(* PLC project Unnamed, Unknown Unnamed 1 *)
(* stored: creationDateTime 2022-08-16T15:49:17, modificationDateTime 2025-06-02T17:15:43 *)

PROGRAM Blink
  VAR
    blink_led : BOOL;
    TON0 : TON;
    TOF0 : TOF;
  END_VAR

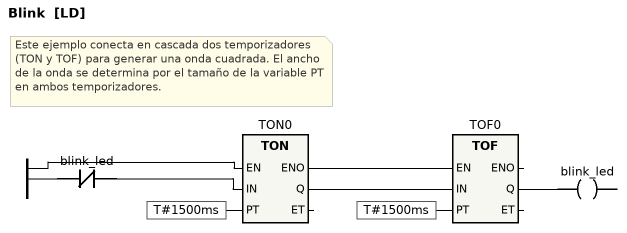
(* LD diagram, written out as Structured Text *)
(* Este ejemplo conecta en cascada dos temporizadores (TON y TOF) para generar una onda cuadrada. El ancho de la onda se determina por el tamaño de la variable PT en ambos temporizadores. *)
TON0(IN := NOT blink_led, PT := T#1500ms);
TOF0(EN := TON0.ENO, IN := TON0.Q, PT := T#1500ms);
blink_led := TOF0.Q;
END_PROGRAM

CONFIGURATION Config0
  RESOURCE Res0 ON PLC
    TASK task0(INTERVAL := T#20ms, PRIORITY := 0);
    PROGRAM instance0 WITH task0 : Blink;
  END_RESOURCE
END_CONFIGURATION
